Staubli VAL3: TRACK.dtx

public Tracks tTraj{}
